# EPICS substitutions: examples/nanodac_absolute/nanodacApp/Db/nanodac.substitutions
file nd.template
{
pattern {S, ND, NI}
	{SECAGE:, SE:ND7B:, 1}
}
